TYPE ST_Sub1 EXTENDS ST_Base1:
STRUCT
	ttime :TIME;
	tton  : TON;
END_STRUCT
END_TYPE

(* stored: Version 1.1.0.1, ProductVersion 3.1.4024.12
   DUT ST_Sub1: Id {287843c4-9e72-4ec0-9b8a-345ce83b6b58} *)
